FUNCTION_BLOCK ProfibusMaster
VAR_INPUT
END_VAR
VAR_OUTPUT
END_VAR
VAR
	Error AT%I* : USINT;
	ActualModulo AT%I* : USINT;
	DiagFlag AT%i* : BOOL;
END_VAR

END_FUNCTION_BLOCK

(* stored: Version 1.1.0.1, ProductVersion 3.1.4024.11
   POU ProfibusMaster: Id {6bceab5d-de58-4a8b-aae3-198c30adc94d}, SpecialFunc None *)
